Staubli VAL3: DataSend2PC.pgx

program DataSend2PC()
  local num jold
  local bool bReconnect
begin
  //this routine is to send the data to PC
  while true
    delay(0)
  endWhile
end
